Fanuc KAREL source: kb00125.KL

-- PROVISIONAL review KL for V1013-1; original PC SHA256 912a8f36b8257758831aae31c2b4c184f5e8650300ccbad970919b4a14439af7
-- Incomplete behavior may be omitted. Consult companion uncertainty JSON. Do not deploy.
PROGRAM KB00125
%NOLOCKGROUP
BEGIN
  -- UNRESOLVED_PC offsets 5-14; opcodes 3F,75
  -- UNRESOLVED_PC offsets 19-26; opcodes 9D,23
  -- UNRESOLVED_PC offsets 31-49; opcodes 27,22,2A,22,31
  -- UNRESOLVED_PC offsets 54-58; opcodes 7F
END KB00125
